TYPE ST_HRErrHist :
STRUCT
{attribute 'displaymode':='hex'}
	hrErrCode	: HRESULT;
	sErrSource	: STRING(63);
	nErrCount	: UDINT;
END_STRUCT
END_TYPE

(* stored: Version 1.1.0.1, ProductVersion 3.1.4024.12
   DUT ST_HRErrHist: Id {92d421d1-d14f-450b-983f-70e2be9df404} *)
